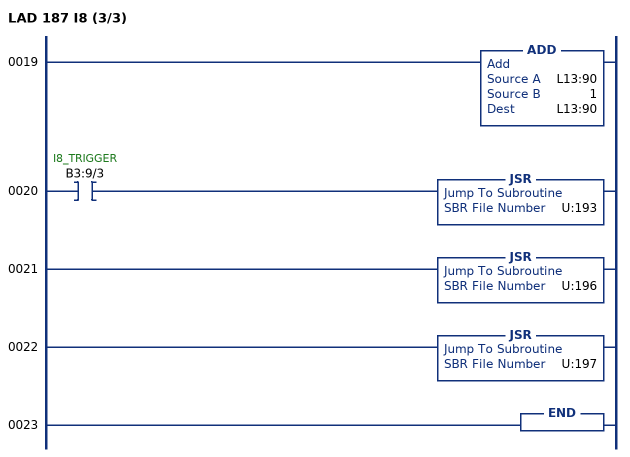
% Rung: 19 %
SOR ADD L13:90 1 L13:90 EOR
% Rung: 20 %
SOR XIC B3:9/3 JSR U:193 EOR
%   B3:9/3  I8_TRIGGER %
% Rung: 21 %
SOR JSR U:196 EOR
% Rung: 22 %
SOR JSR U:197 EOR
% Rung: 23 %
SOR END EOR

LADDER 188 "I8 RESULT"
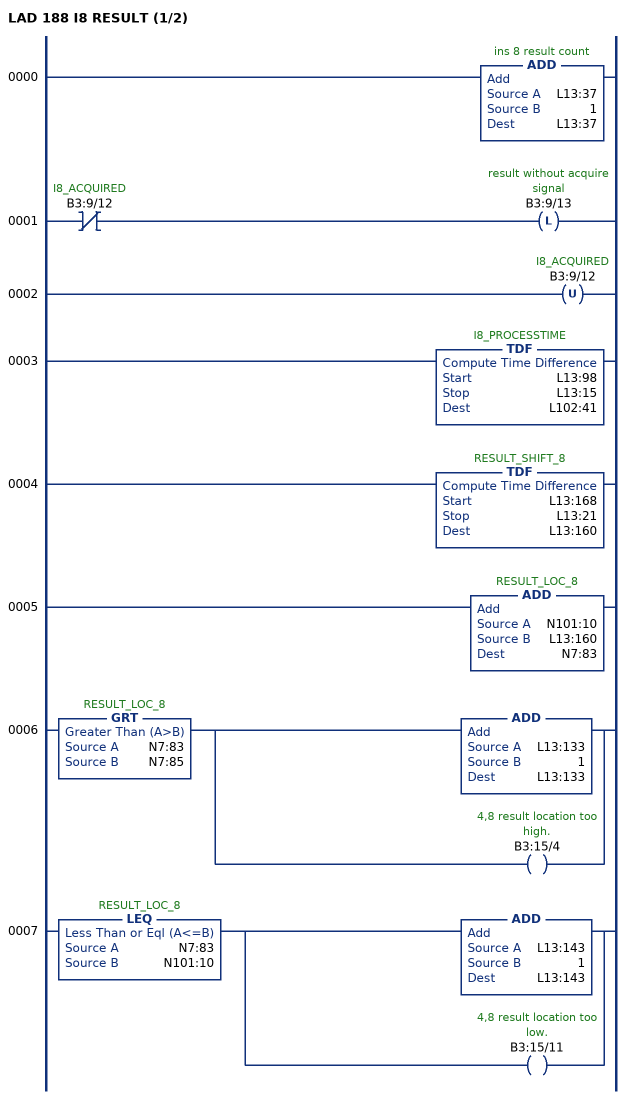
% Rung: 0 %
SOR ADD L13:37 1 L13:37 EOR
%   L13:37  "ins 8 result count" %
% Rung: 1 %
SOR XIO B3:9/12 OTL B3:9/13 EOR
%   B3:9/12  I8_ACQUIRED %
%   B3:9/13  "result without acquire signal" %
% Rung: 2 %
SOR OTU B3:9/12 EOR
%   B3:9/12  I8_ACQUIRED %
% Rung: 3 %
SOR TDF L13:98 L13:15 L102:41 EOR
%   L13:98  I8_TIMEOFACQ %
%   L13:15  THE_TIME %
%   L102:41  I8_PROCESSTIME %
% Rung: 4 %
SOR TDF L13:168 L13:21 L13:160 EOR
%   L13:168  I8_PROCESS_START_POS %
%   L13:21  TOP_POSITION %
%   L13:160  RESULT_SHIFT_8 %
% Rung: 5 %
SOR ADD N101:10 L13:160 N7:83 EOR
%   N101:10  I8_TRIG_LOC %
%   L13:160  RESULT_SHIFT_8 %
%   N7:83  RESULT_LOC_8 %
% Rung: 6 %
SOR GRT N7:83 N7:85 BST ADD L13:133 1 L13:133 NXB OTE B3:15/4 BND EOR
%   N7:83  RESULT_LOC_8 %
%   N7:85  I8_MAX_SHIFT %
%   B3:15/4  "4,8 result location too high." %
% Rung: 7 %
SOR LEQ N7:83 N101:10 BST ADD L13:143 1 L13:143 NXB OTE B3:15/11 BND EOR
%   N7:83  RESULT_LOC_8 %
%   N101:10  I8_TRIG_LOC %
%   B3:15/11  "4,8 result location too low." %

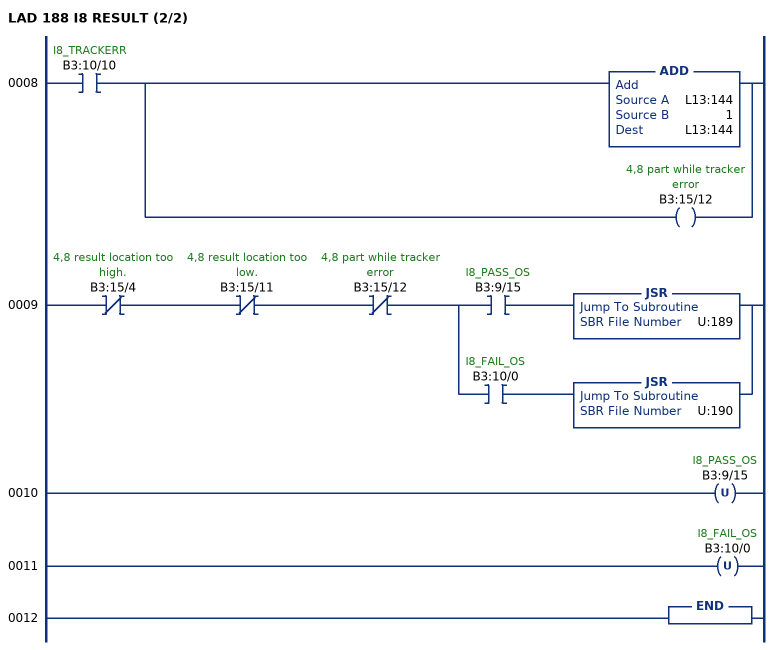
% Rung: 8 %
SOR XIC B3:10/10 BST ADD L13:144 1 L13:144 NXB OTE B3:15/12 BND EOR
%   B3:10/10  I8_TRACKERR %
%   B3:15/12  "4,8 part while tracker error" %
% Rung: 9 %
SOR XIO B3:15/4 XIO B3:15/11 XIO B3:15/12 BST XIC B3:9/15 JSR U:189 NXB XIC B3:10/0 JSR U:190 BND EOR
%   B3:15/4  "4,8 result location too high." %
%   B3:15/11  "4,8 result location too low." %
%   B3:15/12  "4,8 part while tracker error" %
%   B3:9/15  I8_PASS_OS %
%   B3:10/0  I8_FAIL_OS %
% Rung: 10 %
SOR OTU B3:9/15 EOR
%   B3:9/15  I8_PASS_OS %
% Rung: 11 %
SOR OTU B3:10/0 EOR
%   B3:10/0  I8_FAIL_OS %
% Rung: 12 %
SOR END EOR

LADDER 189 "I8 PASS"
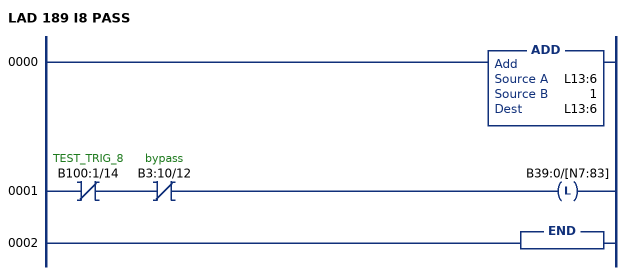
% Rung: 0 %
SOR ADD L13:6 1 L13:6 EOR
% Rung: 1 %
SOR XIO B100:1/14 XIO B3:10/12 OTL B39:0/[N7:83] EOR
%   B100:1/14  TEST_TRIG_8 %
%   B3:10/12  "bypass" %
%   B39:0  TOP_OK_2 %
%   N7:83  RESULT_LOC_8 %
% Rung: 2 %
SOR END EOR

LADDER 190 "I8 FAIL"
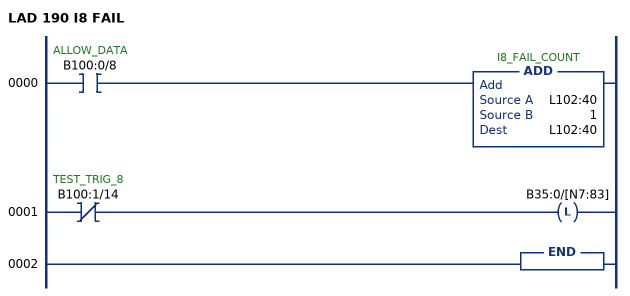
% Rung: 0 %
SOR XIC B100:0/8 ADD L102:40 1 L102:40 EOR
%   B100:0/8  ALLOW_DATA %
%   L102:40  I8_FAIL_COUNT %
% Rung: 1 %
SOR XIO B100:1/14 OTL B35:0/[N7:83] EOR
%   B100:1/14  TEST_TRIG_8 %
%   B35:0  TOP_NG %
%   N7:83  RESULT_LOC_8 %
% Rung: 2 %
SOR END EOR

LADDER 191 "I8 ACQ"
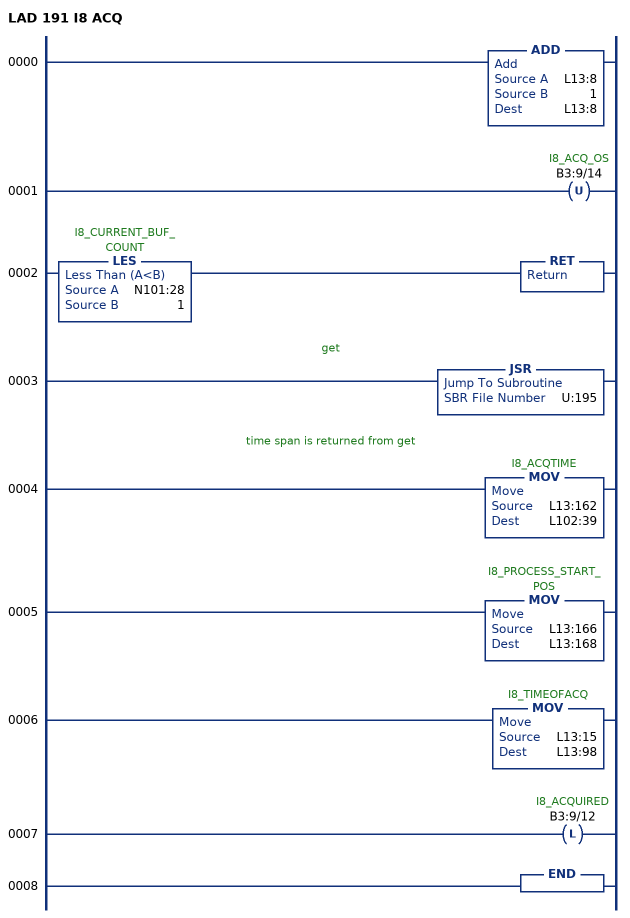
% Rung: 0 %
SOR ADD L13:8 1 L13:8 EOR
% Rung: 1 %
SOR OTU B3:9/14 EOR
%   B3:9/14  I8_ACQ_OS %
% Rung: 2 %
SOR LES N101:28 1 RET EOR
%   N101:28  I8_CURRENT_BUF_COUNT %
% Rung: 3 %
% get %
SOR JSR U:195 EOR
% Rung: 4 %
% time span is returned from get %
SOR MOV L13:162 L102:39 EOR
%   L13:162  I8_TIME_SPAN %
%   L102:39  I8_ACQTIME %
% Rung: 5 %
SOR MOV L13:166 L13:168 EOR
%   L13:166  I8_PULLED_POSITION %
%   L13:168  I8_PROCESS_START_POS %
% Rung: 6 %
SOR MOV L13:15 L13:98 EOR
%   L13:15  THE_TIME %
%   L13:98  I8_TIMEOFACQ %
% Rung: 7 %
SOR OTL B3:9/12 EOR
%   B3:9/12  I8_ACQUIRED %
% Rung: 8 %
SOR END EOR

LADDER 192 "I8 TESTER"
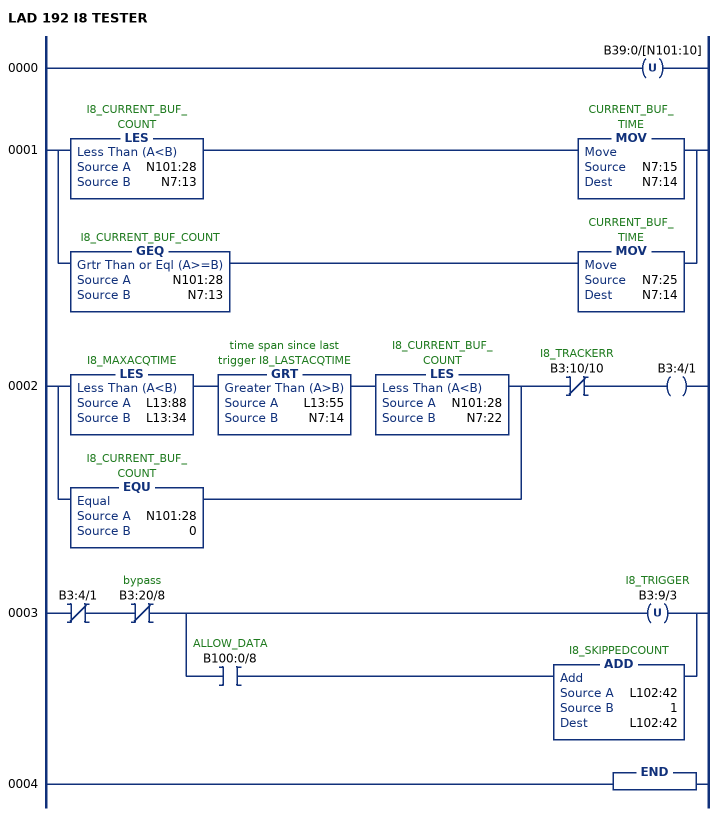
% Rung: 0 %
SOR OTU B39:0/[N101:10] EOR
%   B39:0  TOP_OK_2 %
%   N101:10  I8_TRIG_LOC %
% Rung: 1 %
SOR BST LES N101:28 N7:13 MOV N7:15 N7:14 NXB GEQ N101:28 N7:13 MOV N7:25 N7:14 BND EOR
%   N101:28  I8_CURRENT_BUF_COUNT %
%   N7:13  BUF_TRANS  "cam to pc buf transition" %
%   N7:15  CAM_BUF_TIME  "cam buf time" %
%   N7:14  CURRENT_BUF_TIME %
%   N7:25  PC_BUF_TIME  "pc buf time" %
% Rung: 2 %
SOR BST LES L13:88 L13:34 GRT L13:55 N7:14 LES N101:28 N7:22 NXB EQU N101:28 0 BND XIO B3:10/10 OTE B3:4/1 EOR
%   L13:88  I8_MAXACQTIME %
%   L13:34  MAX_ACQ_ALL  "absolute max acquire time before bypass trigger" %
%   L13:55  I8_LASTACQTIME  "time span since last trigger" %
%   N7:14  CURRENT_BUF_TIME %
%   N101:28  I8_CURRENT_BUF_COUNT %
%   N7:22  MAX_BUF_ALL  "max buffer count alowed before bypass" %
%   B3:10/10  I8_TRACKERR %
% Rung: 3 %
SOR XIO B3:4/1 XIO B3:20/8 BST OTU B3:9/3 NXB XIC B100:0/8 ADD L102:42 1 L102:42 BND EOR
%   B3:20/8  "bypass" %
%   B3:9/3  I8_TRIGGER %
%   B100:0/8  ALLOW_DATA %
%   L102:42  I8_SKIPPEDCOUNT %
% Rung: 4 %
SOR END EOR

LADDER 193 "I8 TRIG"
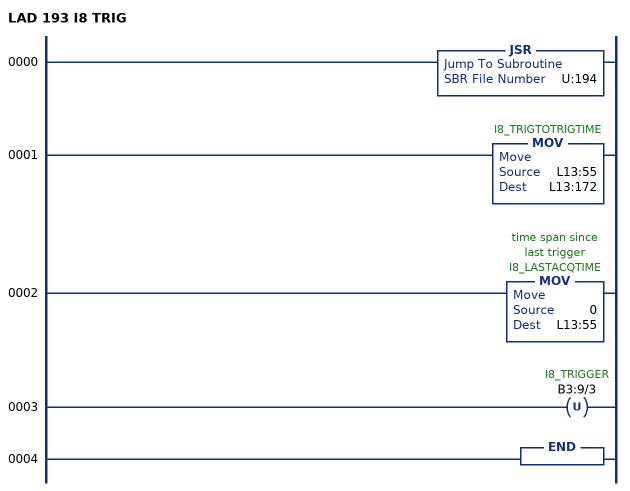
% Rung: 0 %
SOR JSR U:194 EOR
% Rung: 1 %
SOR MOV L13:55 L13:172 EOR
%   L13:55  I8_LASTACQTIME  "time span since last trigger" %
%   L13:172  I8_TRIGTOTRIGTIME %
% Rung: 2 %
SOR MOV 0 L13:55 EOR
%   L13:55  I8_LASTACQTIME  "time span since last trigger" %
% Rung: 3 %
SOR OTU B3:9/3 EOR
%   B3:9/3  I8_TRIGGER %
% Rung: 4 %
SOR END EOR

LADDER 194 "I8 FIFOSET"
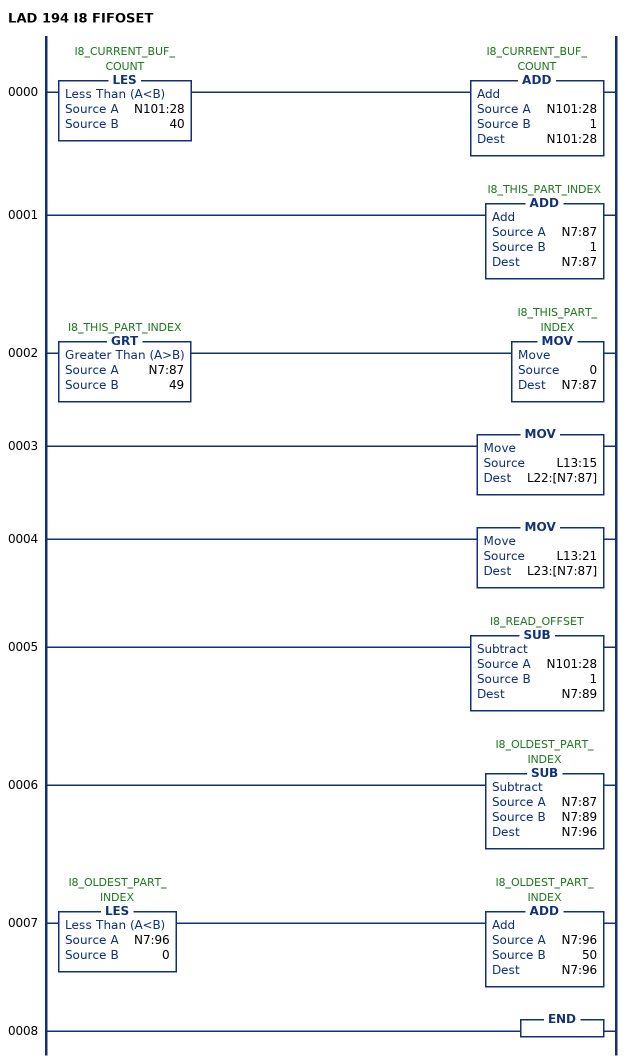
% Rung: 0 %
SOR LES N101:28 40 ADD N101:28 1 N101:28 EOR
%   N101:28  I8_CURRENT_BUF_COUNT %
% Rung: 1 %
SOR ADD N7:87 1 N7:87 EOR
%   N7:87  I8_THIS_PART_INDEX %
% Rung: 2 %
SOR GRT N7:87 49 MOV 0 N7:87 EOR
%   N7:87  I8_THIS_PART_INDEX %
% Rung: 3 %
SOR MOV L13:15 L22:[N7:87] EOR
%   L13:15  THE_TIME %
%   N7:87  I8_THIS_PART_INDEX %
% Rung: 4 %
SOR MOV L13:21 L23:[N7:87] EOR
%   L13:21  TOP_POSITION %
%   N7:87  I8_THIS_PART_INDEX %
% Rung: 5 %
SOR SUB N101:28 1 N7:89 EOR
%   N101:28  I8_CURRENT_BUF_COUNT %
%   N7:89  I8_READ_OFFSET %
% Rung: 6 %
SOR SUB N7:87 N7:89 N7:96 EOR
%   N7:87  I8_THIS_PART_INDEX %
%   N7:89  I8_READ_OFFSET %
%   N7:96  I8_OLDEST_PART_INDEX %
% Rung: 7 %
SOR LES N7:96 0 ADD N7:96 50 N7:96 EOR
%   N7:96  I8_OLDEST_PART_INDEX %
% Rung: 8 %
SOR END EOR

LADDER 195 "I8 FIFOGET"
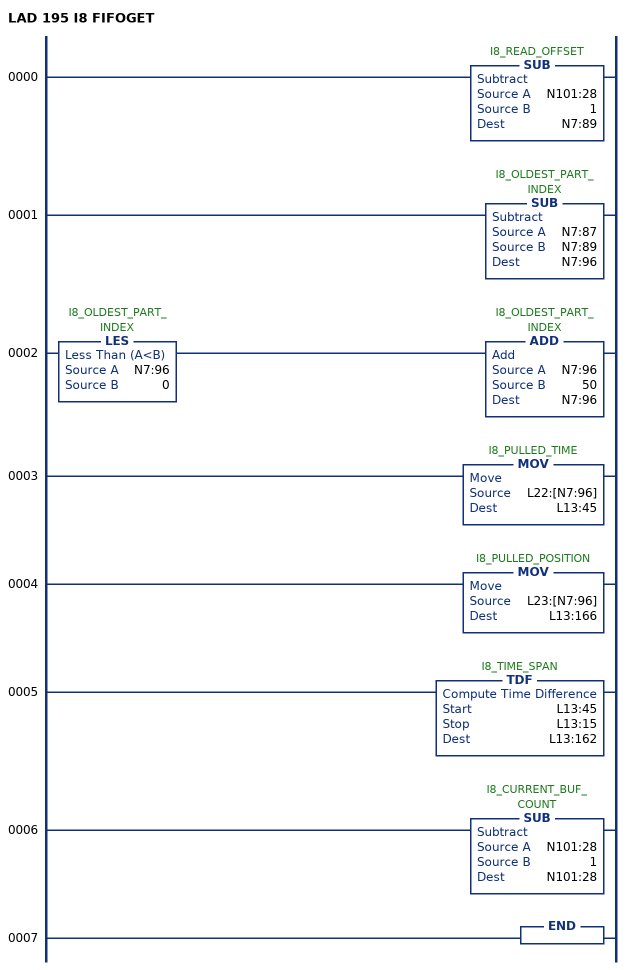
% Rung: 0 %
SOR SUB N101:28 1 N7:89 EOR
%   N101:28  I8_CURRENT_BUF_COUNT %
%   N7:89  I8_READ_OFFSET %
% Rung: 1 %
SOR SUB N7:87 N7:89 N7:96 EOR
%   N7:87  I8_THIS_PART_INDEX %
%   N7:89  I8_READ_OFFSET %
%   N7:96  I8_OLDEST_PART_INDEX %
% Rung: 2 %
SOR LES N7:96 0 ADD N7:96 50 N7:96 EOR
%   N7:96  I8_OLDEST_PART_INDEX %
% Rung: 3 %
SOR MOV L22:[N7:96] L13:45 EOR
%   N7:96  I8_OLDEST_PART_INDEX %
%   L13:45  I8_PULLED_TIME %
% Rung: 4 %
SOR MOV L23:[N7:96] L13:166 EOR
%   N7:96  I8_OLDEST_PART_INDEX %
%   L13:166  I8_PULLED_POSITION %
% Rung: 5 %
SOR TDF L13:45 L13:15 L13:162 EOR
%   L13:45  I8_PULLED_TIME %
%   L13:15  THE_TIME %
%   L13:162  I8_TIME_SPAN %
% Rung: 6 %
SOR SUB N101:28 1 N101:28 EOR
%   N101:28  I8_CURRENT_BUF_COUNT %
% Rung: 7 %
SOR END EOR

LADDER 196 "I8 DATA"
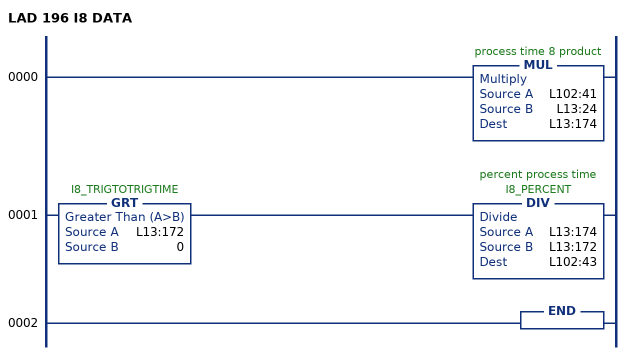
% Rung: 0 %
SOR MUL L102:41 L13:24 L13:174 EOR
%   L102:41  I8_PROCESSTIME %
%   L13:24  "multiplyer to make devision come out to a percentage" %
%   L13:174  "process time 8 product" %
% Rung: 1 %
SOR GRT L13:172 0 DIV L13:174 L13:172 L102:43 EOR
%   L13:172  I8_TRIGTOTRIGTIME %
%   L13:174  "process time 8 product" %
%   L102:43  I8_PERCENT  "percent process time" %
% Rung: 2 %
SOR END EOR

LADDER 197 "I8 FAULT"
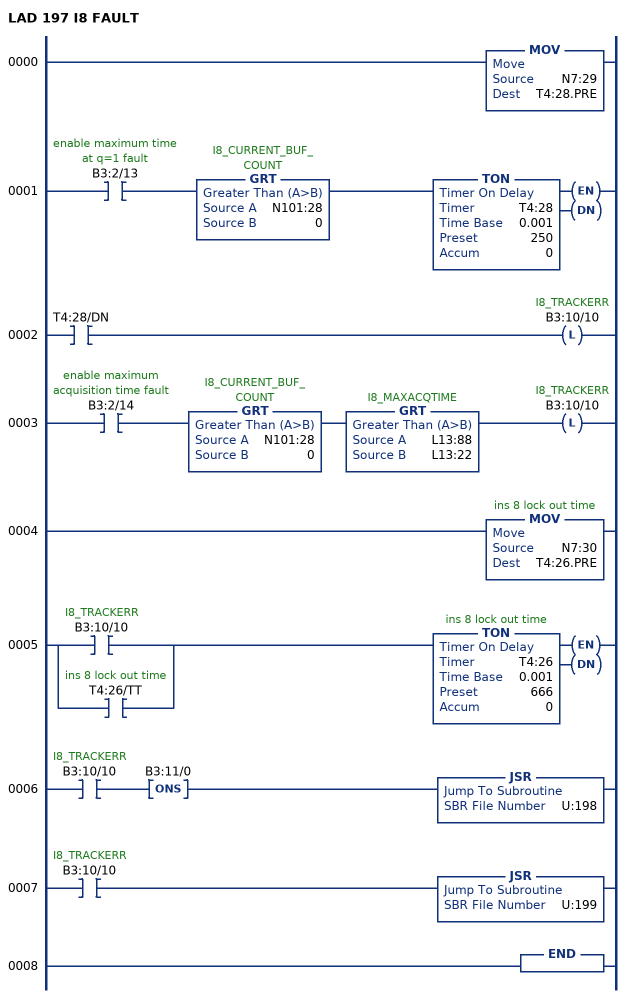
% Rung: 0 %
SOR MOV N7:29 T4:28.PRE EOR
%   N7:29  "max allowed ms time for q to be above 1 if safe fault is used" %
% Rung: 1 %
SOR XIC B3:2/13 GRT N101:28 0 TON T4:28 0.001 250 0 EOR
%   B3:2/13  "enable maximum time at q=1 fault" %
%   N101:28  I8_CURRENT_BUF_COUNT %
% Rung: 2 %
SOR XIC T4:28/DN OTL B3:10/10 EOR
%   B3:10/10  I8_TRACKERR %
% Rung: 3 %
SOR XIC B3:2/14 GRT N101:28 0 GRT L13:88 L13:22 OTL B3:10/10 EOR
%   B3:2/14  "enable maximum acquisition time fault" %
%   N101:28  I8_CURRENT_BUF_COUNT %
%   L13:88  I8_MAXACQTIME %
%   L13:22  "maximum of the longest acquire time allowed if maximum acquire time fault is enabled" %
%   B3:10/10  I8_TRACKERR %
% Rung: 4 %
SOR MOV N7:30 T4:26.PRE EOR
%   N7:30  "ms time setting to lock out inspection to give all pending images a chance to clear" %
%   T4:26  "ins 8 lock out time" %
% Rung: 5 %
SOR BST XIC B3:10/10 NXB XIC T4:26/TT BND TON T4:26 0.001 666 0 EOR
%   B3:10/10  I8_TRACKERR %
%   T4:26  "ins 8 lock out time" %
% Rung: 6 %
SOR XIC B3:10/10 ONS B3:11/0 JSR U:198 EOR
%   B3:10/10  I8_TRACKERR %
% Rung: 7 %
SOR XIC B3:10/10 JSR U:199 EOR
%   B3:10/10  I8_TRACKERR %
% Rung: 8 %
SOR END EOR

LADDER 198 "I8 FIX1"
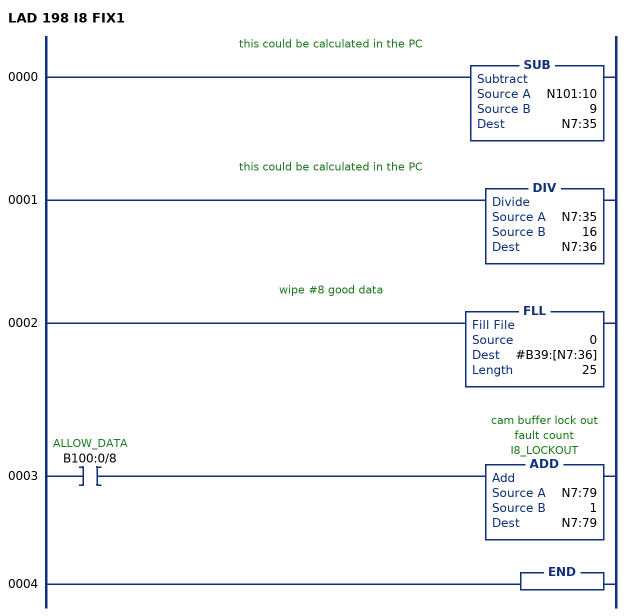
% Rung: 0 %
% this could be calculated in the PC %
SOR SUB N101:10 9 N7:35 EOR
%   N101:10  I8_TRIG_LOC %
% Rung: 1 %
% this could be calculated in the PC %
SOR DIV N7:35 16 N7:36 EOR
% Rung: 2 %
% wipe #8 good data %
SOR FLL 0 #B39:[N7:36] 25 EOR
% Rung: 3 %
SOR XIC B100:0/8 ADD N7:79 1 N7:79 EOR
%   B100:0/8  ALLOW_DATA %
%   N7:79  I8_LOCKOUT  "cam buffer lock out fault count" %
% Rung: 4 %
SOR END EOR

LADDER 199 "I8 FIX2"
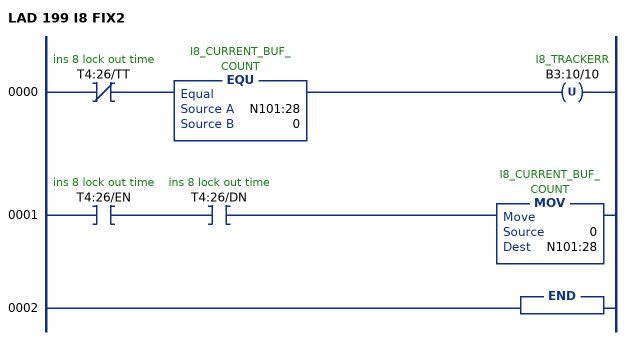
% Rung: 0 %
SOR XIO T4:26/TT EQU N101:28 0 OTU B3:10/10 EOR
%   T4:26  "ins 8 lock out time" %
%   N101:28  I8_CURRENT_BUF_COUNT %
%   B3:10/10  I8_TRACKERR %
% Rung: 1 %
SOR XIC T4:26/EN XIC T4:26/DN MOV 0 N101:28 EOR
%   T4:26  "ins 8 lock out time" %
%   N101:28  I8_CURRENT_BUF_COUNT %
% Rung: 2 %
SOR END EOR

LADDER 200 "PASS BLOW"
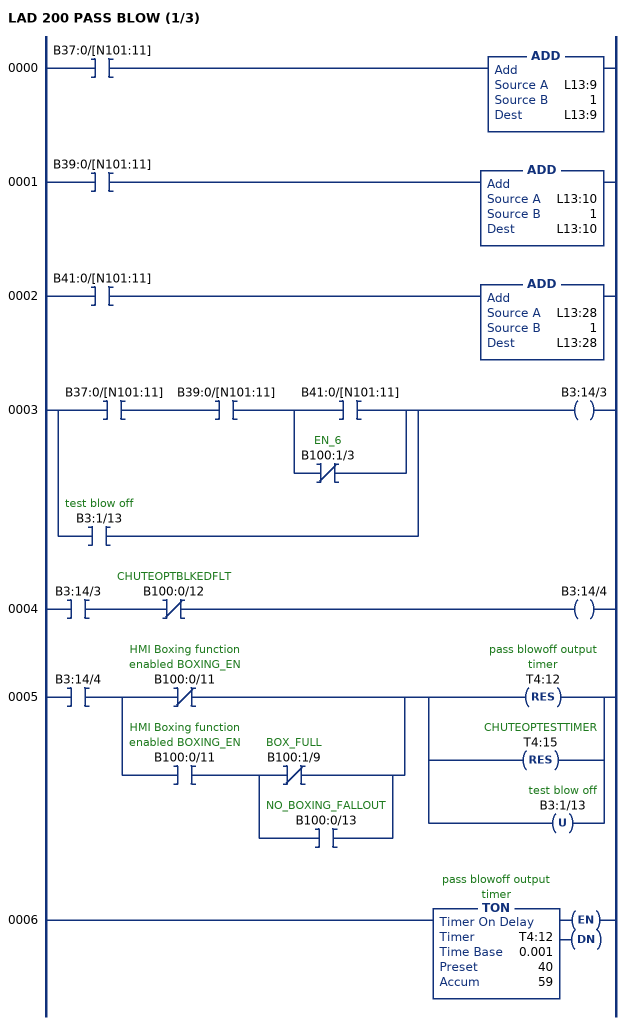
% Rung: 0 %
SOR XIC B37:0/[N101:11] ADD L13:9 1 L13:9 EOR
%   B37:0  TOP_OK_1 %
%   N101:11  BLOW_PT %
% Rung: 1 %
SOR XIC B39:0/[N101:11] ADD L13:10 1 L13:10 EOR
%   B39:0  TOP_OK_2 %
%   N101:11  BLOW_PT %
% Rung: 2 %
SOR XIC B41:0/[N101:11] ADD L13:28 1 L13:28 EOR
%   B41:0  TOP_OK_3 %
%   N101:11  BLOW_PT %
% Rung: 3 %
SOR BST XIC B37:0/[N101:11] XIC B39:0/[N101:11] BST XIC B41:0/[N101:11] NXB XIO B100:1/3 BND NXB XIC B3:1/13 BND OTE B3:14/3 EOR
%   B37:0  TOP_OK_1 %
%   N101:11  BLOW_PT %
%   B39:0  TOP_OK_2 %
%   B41:0  TOP_OK_3 %
%   B100:1/3  EN_6 %
%   B3:1/13  "test blow off" %
% Rung: 4 %
SOR XIC B3:14/3 XIO B100:0/12 OTE B3:14/4 EOR
%   B100:0/12  CHUTEOPTBLKEDFLT %
% Rung: 5 %
SOR XIC B3:14/4 BST XIO B100:0/11 NXB XIC B100:0/11 BST XIO B100:1/9 NXB XIC B100:0/13 BND BND BST RES T4:12 NXB RES T4:15 NXB OTU B3:1/13 BND EOR
%   B100:0/11  BOXING_EN  "HMI Boxing function enabled" %
%   B100:1/9  BOX_FULL %
%   B100:0/13  NO_BOXING_FALLOUT %
%   T4:12  "pass blowoff output timer" %
%   T4:15  CHUTEOPTESTTIMER %
%   B3:1/13  "test blow off" %
% Rung: 6 %
SOR TON T4:12 0.001 40 59 EOR
%   T4:12  "pass blowoff output timer" %

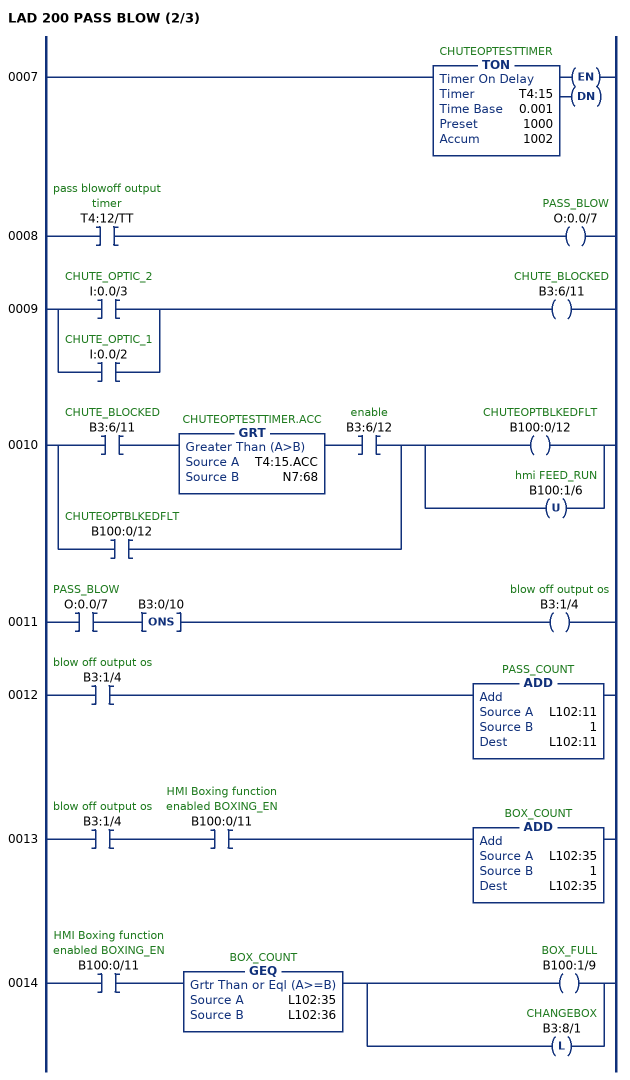
% Rung: 7 %
SOR TON T4:15 0.001 1000 1002 EOR
%   T4:15  CHUTEOPTESTTIMER %
% Rung: 8 %
SOR XIC T4:12/TT OTE O:0.0/7 EOR
%   T4:12  "pass blowoff output timer" %
%   O:0.0/7  PASS_BLOW %
% Rung: 9 %
SOR BST XIC I:0.0/3 NXB XIC I:0.0/2 BND OTE B3:6/11 EOR
%   I:0.0/3  CHUTE_OPTIC_2 %
%   I:0.0/2  CHUTE_OPTIC_1 %
%   B3:6/11  CHUTE_BLOCKED %
% Rung: 10 %
SOR BST XIC B3:6/11 GRT T4:15.ACC N7:68 XIC B3:6/12 NXB XIC B100:0/12 BND BST OTE B100:0/12 NXB OTU B100:1/6 BND EOR
%   B3:6/11  CHUTE_BLOCKED %
%   T4:15  CHUTEOPTESTTIMER %
%   B3:6/12  "enable" %
%   B100:0/12  CHUTEOPTBLKEDFLT %
%   B100:1/6  FEED_RUN  "hmi" %
% Rung: 11 %
SOR XIC O:0.0/7 ONS B3:0/10 OTE B3:1/4 EOR
%   O:0.0/7  PASS_BLOW %
%   B3:1/4  "blow off output os" %
% Rung: 12 %
SOR XIC B3:1/4 ADD L102:11 1 L102:11 EOR
%   B3:1/4  "blow off output os" %
%   L102:11  PASS_COUNT %
% Rung: 13 %
SOR XIC B3:1/4 XIC B100:0/11 ADD L102:35 1 L102:35 EOR
%   B3:1/4  "blow off output os" %
%   B100:0/11  BOXING_EN  "HMI Boxing function enabled" %
%   L102:35  BOX_COUNT %
% Rung: 14 %
SOR XIC B100:0/11 GEQ L102:35 L102:36 BST OTE B100:1/9 NXB OTL B3:8/1 BND EOR
%   B100:0/11  BOXING_EN  "HMI Boxing function enabled" %
%   L102:35  BOX_COUNT %
%   L102:36  BOX_LIMIT  "box count setpoint" %
%   B100:1/9  BOX_FULL %
%   B3:8/1  CHANGEBOX %

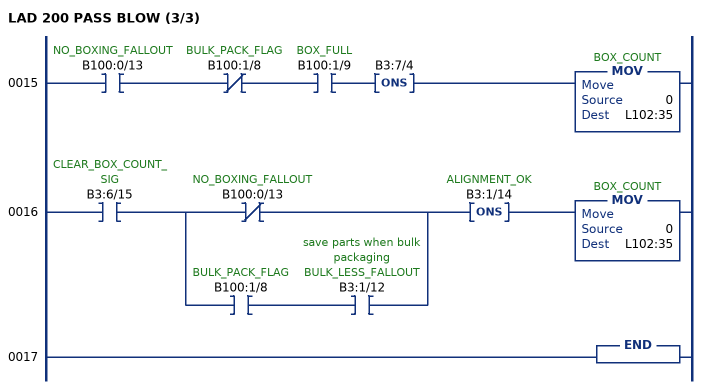
% Rung: 15 %
SOR XIC B100:0/13 XIO B100:1/8 XIC B100:1/9 ONS B3:7/4 MOV 0 L102:35 EOR
%   B100:0/13  NO_BOXING_FALLOUT %
%   B100:1/8  BULK_PACK_FLAG %
%   B100:1/9  BOX_FULL %
%   L102:35  BOX_COUNT %
% Rung: 16 %
SOR XIC B3:6/15 BST XIO B100:0/13 NXB XIC B100:1/8 XIC B3:1/12 BND ONS B3:1/14 MOV 0 L102:35 EOR
%   B3:6/15  CLEAR_BOX_COUNT_SIG %
%   B100:0/13  NO_BOXING_FALLOUT %
%   B100:1/8  BULK_PACK_FLAG %
%   B3:1/12  BULK_LESS_FALLOUT  "save parts when bulk packaging" %
%   B3:1/14  ALIGNMENT_OK %
%   L102:35  BOX_COUNT %
% Rung: 17 %
SOR END EOR

LADDER 235 "TESTTRIGS"    % highspeed test triggers, not necessary %
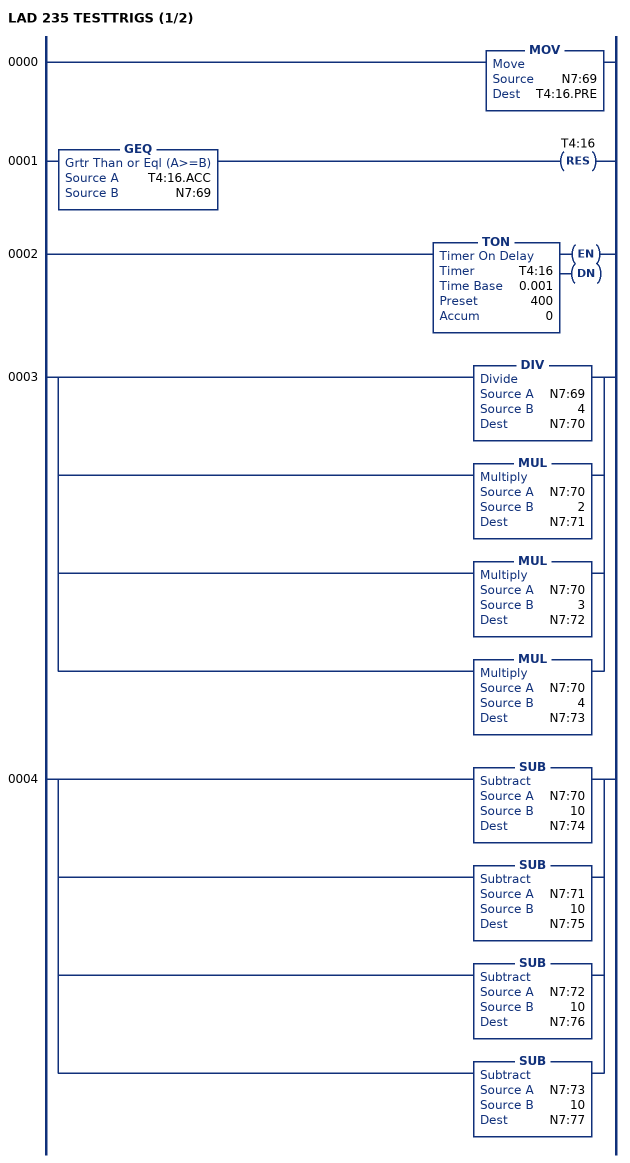
% Rung: 0 %
SOR MOV N7:69 T4:16.PRE EOR
% Rung: 1 %
SOR GEQ T4:16.ACC N7:69 RES T4:16 EOR
% Rung: 2 %
SOR TON T4:16 0.001 400 0 EOR
% Rung: 3 %
SOR BST DIV N7:69 4 N7:70 NXB MUL N7:70 2 N7:71 NXB MUL N7:70 3 N7:72 NXB MUL N7:70 4 N7:73 BND EOR
% Rung: 4 %
SOR BST SUB N7:70 10 N7:74 NXB SUB N7:71 10 N7:75 NXB SUB N7:72 10 N7:76 NXB SUB N7:73 10 N7:77 BND EOR

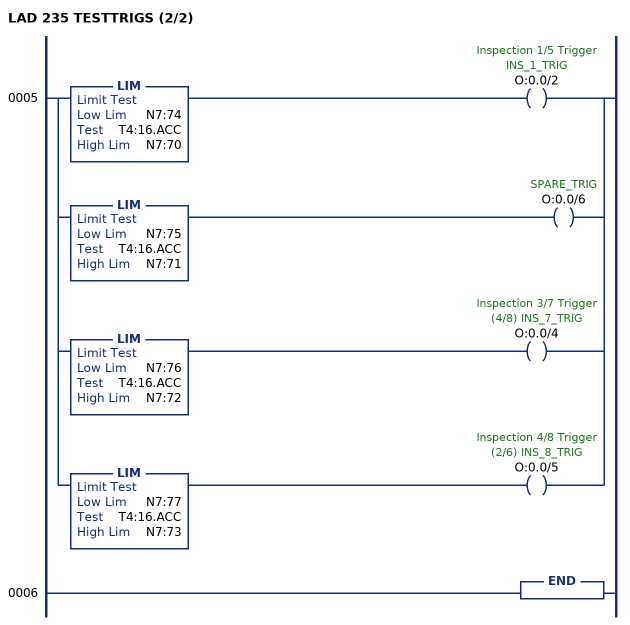
% Rung: 5 %
SOR BST LIM N7:74 T4:16.ACC N7:70 OTE O:0.0/2 NXB LIM N7:75 T4:16.ACC N7:71 OTE O:0.0/6 NXB LIM N7:76 T4:16.ACC N7:72 OTE O:0.0/4 NXB LIM N7:77 T4:16.ACC N7:73 OTE O:0.0/5 BND EOR
%   O:0.0/2  INS_1_TRIG  "Inspection 1/5 Trigger" %
%   O:0.0/6  SPARE_TRIG %
%   O:0.0/4  INS_7_TRIG  "Inspection 3/7 Trigger (4/8)" %
%   O:0.0/5  INS_8_TRIG  "Inspection 4/8 Trigger (2/6)" %
% Rung: 6 %
SOR END EOR

LADDER 236 "TESTTRIG1"
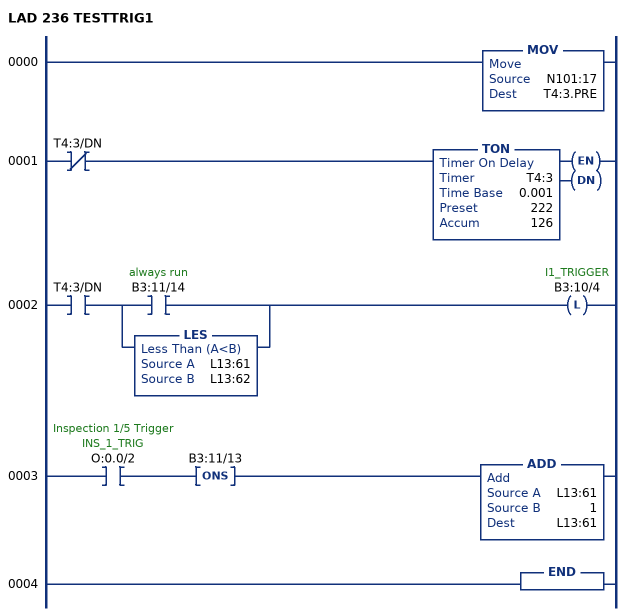
% Rung: 0 %
SOR MOV N101:17 T4:3.PRE EOR
%   N101:17  I1_TRIGTIME  "test trigger 1 interval" %
% Rung: 1 %
SOR XIO T4:3/DN TON T4:3 0.001 222 126 EOR
% Rung: 2 %
SOR XIC T4:3/DN BST XIC B3:11/14 NXB LES L13:61 L13:62 BND OTL B3:10/4 EOR
%   B3:11/14  "always run" %
%   B3:10/4  I1_TRIGGER %
% Rung: 3 %
SOR XIC O:0.0/2 ONS B3:11/13 ADD L13:61 1 L13:61 EOR
%   O:0.0/2  INS_1_TRIG  "Inspection 1/5 Trigger" %
% Rung: 4 %
SOR END EOR

LADDER 237 "TESTTRIG2"
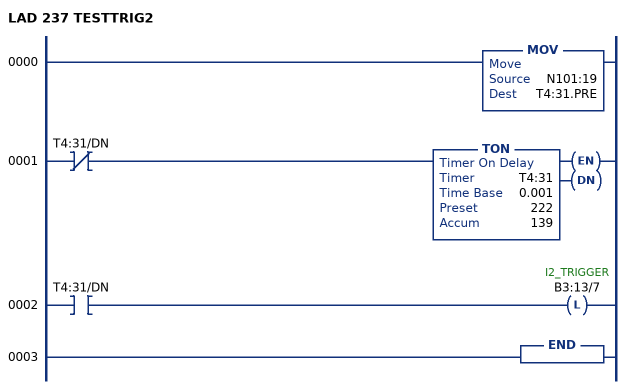
% Rung: 0 %
SOR MOV N101:19 T4:31.PRE EOR
%   N101:19  I2_I6_TRIGTIME  "test trgiger 2/6 interval" %
% Rung: 1 %
SOR XIO T4:31/DN TON T4:31 0.001 222 139 EOR
% Rung: 2 %
SOR XIC T4:31/DN OTL B3:13/7 EOR
%   B3:13/7  I2_TRIGGER %
% Rung: 3 %
SOR END EOR

LADDER 238 "TESTTRIG3"
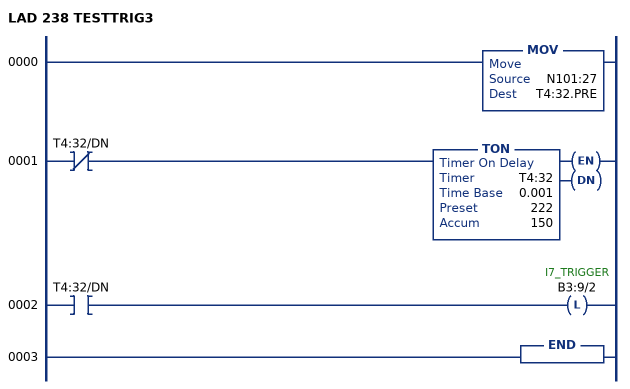
% Rung: 0 %
SOR MOV N101:27 T4:32.PRE EOR
%   N101:27  I7_TRIGTIME %
% Rung: 1 %
SOR XIO T4:32/DN TON T4:32 0.001 222 150 EOR
% Rung: 2 %
SOR XIC T4:32/DN OTL B3:9/2 EOR
%   B3:9/2  I7_TRIGGER %
% Rung: 3 %
SOR END EOR

LADDER 239 "TESTTRIG4"
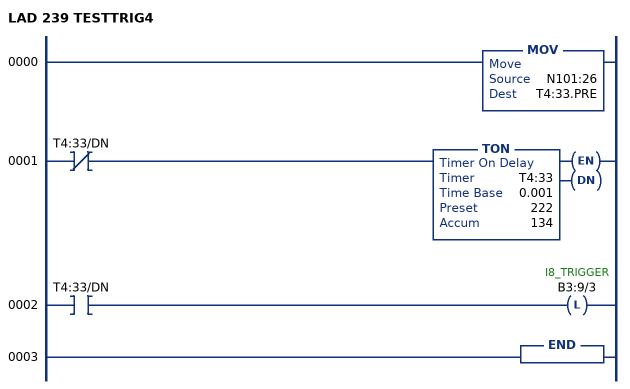
% Rung: 0 %
SOR MOV N101:26 T4:33.PRE EOR
%   N101:26  I8_TRIGTIME %
% Rung: 1 %
SOR XIO T4:33/DN TON T4:33 0.001 222 134 EOR
% Rung: 2 %
SOR XIC T4:33/DN OTL B3:9/3 EOR
%   B3:9/3  I8_TRIGGER %
% Rung: 3 %
SOR END EOR

LADDER 240 "TESTTRIG5"
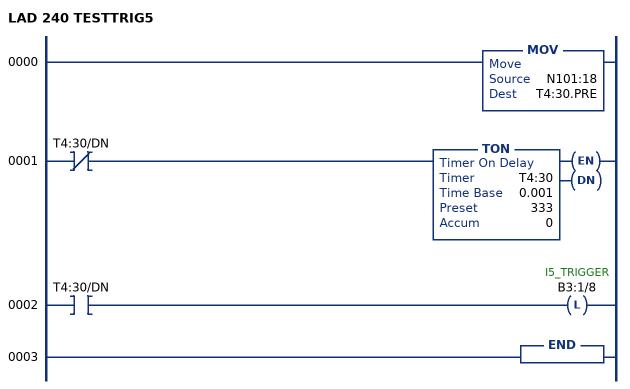
% Rung: 0 %
SOR MOV N101:18 T4:30.PRE EOR
%   N101:18  I5_TRIGTIME  "test trigger 5 interval" %
% Rung: 1 %
SOR XIO T4:30/DN TON T4:30 0.001 333 0 EOR
% Rung: 2 %
SOR XIC T4:30/DN OTL B3:1/8 EOR
%   B3:1/8  I5_TRIGGER %
% Rung: 3 %
SOR END EOR

LADDER 241 "TESTTRIG6"
